FUNCTION F_LH_SV : STRING
VAR_INPUT
	SV: REAL;
	nDecimal: INT := 0;
END_VAR
VAR
	iPV: INT;
	wPV: WORD;
	i: INT;
	r1: REAL;
END_VAR


r1 := SV;

//Decimal
FOR i := 0 TO nDecimal - 1 BY 1 DO
	r1 := r1 * 10;
END_FOR

iPV := REAL_TO_INT(r1);
wPV := INT_TO_WORD(iPV);

F_LH_SV := WORD_TO_HEXSTR(in:= wPV, iPrecision:= 4, bLoCase:= FALSE);

END_FUNCTION

(* stored: Version 1.1.0.1, ProductVersion 3.1.4024.12
   POU F_LH_SV: Id {64045691-07f5-48f9-8321-3c4d0796b468}, SpecialFunc None *)
